PROGRAM S14_LabelChecking
VAR
	//工站
	station					: REFERENCE TO FB_Station:=fbstation[14];
	
//气缸
	fbHOZCyl_1			:REFERENCE TO FB_Cylinder:=fbCylinder[37];	//	推料气缸1
	fbHOZCyl_2			:REFERENCE TO FB_Cylinder:=fbCylinder[38];	//	推料气缸2
	
	//延时
	arTonDelay :ARRAY[1..20] OF TON;
	//返回值
	UdiReturnValue :ARRAY[1..20] OF UDINT;
	
	
	
	i: INT;

END_VAR

A_Input();
Alarm();
Delay();
FlowAuto();
FlowInit();
General();
ILC();
TipAuto();
TipManual();
Z_Output();

ACTION A_Input:
//气缸
fbHOZCyl_1.xWP_Sensor:=					IxS12HOZCyl_1WP;//	贴标检测工位¶推料气缸1¶动点
fbHOZCyl_1.xHP_Sensor:=					IxS12HOZCyl_1HP;//	贴标检测工位¶推料气缸1¶原点
fbHOZCyl_2.xWP_Sensor:=					IxS12HOZCyl_2WP;//	贴标检测工位¶推料气缸2¶动点
fbHOZCyl_2.xHP_Sensor:=					IxS12HOZCyl_2HP;//	贴标检测工位¶推料气缸2¶原点
END_ACTION

ACTION Alarm:
//
station.adwAlarm[1].00:=station.xInitTimeout;	  			//S08Label 初始化超时
END_ACTION

ACTION Delay:
(*arTonDelay[01](IN:= , PT:=T#0.1S , Q=> , ET=> );*)//TipAuto使用
arTonDelay[02](IN:=  , PT:=T#1S , Q=> , ET=> );
arTonDelay[03](IN:=   , PT:=T#1S , Q=> , ET=> );
arTonDelay[04](IN:= , PT:=T#0.1S , Q=> , ET=> );
arTonDelay[05](IN:= , PT:=T#0.1S , Q=> , ET=> );
arTonDelay[06](IN:= , PT:=T#0.1S , Q=> , ET=> );
arTonDelay[07](IN:= , PT:=T#0.1S , Q=> , ET=> );
arTonDelay[08](IN:= , PT:=T#0.1S , Q=> , ET=> );
arTonDelay[09](IN:= , PT:=T#0.1S , Q=> , ET=> );
END_ACTION

ACTION FlowAuto:

//-----------------------------------------初始化是否完成判断----------------------------------------------
IF NOT station.xInitDone 
THEN
 	station.iStepAuto:=0;
 	station.xDone:=FALSE;
	station.xRunningOffProhibit := FALSE ;//运行中信号Off禁止
ELSIF station.xRunning  OR   station.xRunningOffProhibit
THEN
//-----------------------------------------动作步骤--------------------------------------------------------
CASE station.iStepAuto OF	  
	0: //----Home Step，等待启动----
		IF station.xDisabled 
			AND station.xCanRun 
			AND NOT fbMachine[1].xStopped 
			AND NOT station.xSingleRunning 
		THEN
			station.xDone:=TRUE;
		END_IF
		
		IF  station.xSingleRunning 
			OR station.xCanRun 
			AND NOT station.xDone 
			AND NOT station.xDisabled 
			AND NOT fbMachine[1].xStopped
		THEN
			station.xCycleEnable:=TRUE;
			station.xDone:= FALSE;  
			station.xRunningOffProhibit := TRUE ;//运行中信号Off禁止
			station.iStepAuto:= 10;
		END_IF
    10: //复位数据 
			station.iStepAuto:=20;

	
	999://----Single Run Finish----
			
		station.iStepAuto :=0;
		IF NOT station.xSingleContinuousRun THEN
			station.xSingleRunFlag:=FALSE;
		END_IF
		
		station.xCycleEnable:=FALSE;	
		station.xDone:=TRUE;
		station.xRunningOffProhibit := FALSE ;//运行中信号Off禁止
	ELSE
		;	
END_CASE



END_IF
END_ACTION

ACTION FlowInit:
IF NOT station.xIniting THEN
  station.iStepInit:=0;    
ELSE
//--------------------------------------------初始化步序----------------------------------
CASE station.iStepInit OF	
 0://  
  	IF station.xIniting THEN	
  	  station.iStepInit:=10;	
  	END_IF	
10://复位数据
    station.iStepInit:=999;	
999://初始化完成	
	station.iStepInit:=0;
	station.xInitDone:=TRUE;  
END_CASE
END_IF
END_ACTION

ACTION General:

END_ACTION

ACTION ILC:

//---------------------------------------------------工站可执行-------------------------------------------------------
station.xCanRun :=TRUE ;

//---------------------------------------------------气缸动作条件-------------------------------------------
fbHOZCyl_1.xOffILC	:=	TRUE	;
fbHOZCyl_1.xOnILC	:=	TRUE; 

fbHOZCyl_2.xOffILC	:=	TRUE	;
fbHOZCyl_2.xOnILC	:=	TRUE; 


//---------------------------------------------------伺服动作条件-------------------------------------------
END_ACTION

ACTION TipAuto:

//------------------------------------------------AutoTip Cylinder--------------------------------
	
//------------------------------------------------AutoTip Servo--------------------------------
//**************************************
END_ACTION

ACTION TipManual:
//--------------------------------------------ManualTip------------------------------------------------------

//-------------------------------------------气缸提示---------------------------------------------------------




/////////////////////////////////////////////////////////////////////////////////////////////////////////////////
END_ACTION

ACTION Z_Output:
(**************************气缸输出********************************)
QxS12HOZCyl_1WP	:=fbHOZCyl_1.xWP_Valve;//	贴标检测工位¶推料气缸1¶动点
QxS12HOZCyl_1HP	:=fbHOZCyl_1.xHP_Valve;//	贴标检测工位¶推料气缸1¶原点
QxS12HOZCyl_2WP	:=fbHOZCyl_2.xWP_Valve;//	贴标检测工位¶推料气缸2¶动点
QxS12HOZCyl_2HP	:=fbHOZCyl_2.xHP_Valve;//	贴标检测工位¶推料气缸2¶原点
END_ACTION

END_PROGRAM

(* stored: Version 1.1.0.1, ProductVersion 3.1.4024.9
   POU S14_LabelChecking: Id {de280412-b784-48ff-b9e4-45ab603ab4a3}, SpecialFunc None
   Action A_Input: Id {56ab53d4-cea4-4110-a800-d493a02bd0e3}
   Action Alarm: Id {fcf10fe8-b45b-4f97-aec1-69d4e3dfa417}
   Action Delay: Id {7bc9ee60-9b9c-4a53-b951-82315c5dc169}
   Action FlowAuto: Id {8d9b9938-1bf2-4828-8e60-c95a62abe4d7}
   Action FlowInit: Id {35086538-cb4c-4ee9-b035-5fd976ee42d9}
   Action General: Id {4e5f5ae7-ceae-48cf-bdf4-41d615a5187b}
   Action ILC: Id {dd4987fb-dc61-471e-a124-46223fbf39d1}
   Action TipAuto: Id {b36dece4-89a1-4636-a437-523951c4d470}
   Action TipManual: Id {1ef57cb0-c9a2-486b-9130-6b768818a287}
   Action Z_Output: Id {c52e7128-5f2e-405f-a9f7-d94ed1c780d1} *)
